FUNCTION_BLOCK FB_CappingCommand

VAR_INPUT
  IbTrigger                                 : BOOL;
  IbReset                                   : BOOL;
END_VAR

VAR_OUTPUT
  ObCappingCommand                          : BOOL;
END_VAR

VAR
  fb_TonTrigger                             : TON;
  fb_TonReset                               : TON;
  bL_CappingCommandAfterEngaged             : BOOL;
END_VAR

VAR CONSTANT
  tC_DELAY_CAPPING_COMMAND                  : TIME := T#500MS;    (*Delay for automatic generated capping commands*)
  tC_RELEASE_CAPPING_COMMAND                : TIME := T#2S;       (*Release for automatic generated capping commands*)
END_VAR

fb_TonTrigger(IN := IbTrigger, PT := tC_DELAY_CAPPING_COMMAND);
IF fb_TonTrigger.Q THEN
  ObCappingCommand := TRUE;
END_IF
fb_TonReset(IN := IbTrigger, PT := tC_RELEASE_CAPPING_COMMAND);
IF fb_TonReset.Q OR IbReset THEN
  ObCappingCommand := FALSE;
END_IF

END_FUNCTION_BLOCK

(* stored: Version 1.1.0.1, ProductVersion 3.1.4024.9
   POU FB_CappingCommand: Id {a0d6bc23-549b-4287-b93d-e326bc78c1b3}, SpecialFunc None *)
